// TIA Portal V18 export
// export: Created 2025-12-01T17:52:56.9110374Z, ExportSetting None, DisplayName Totally Integrated Automation Portal, DisplayVersion V18 Update 5, DisplayName TIA Portal Openness, DisplayVersion V18 Update 5, DisplayName TIA Portal Teamcenter Gateway, DisplayVersion V18, DisplayName TIA Portal Version Control Interface, DisplayVersion V18, DisplayName STEP 7 Professional, DisplayVersion V18 Update 5, DisplayName STEP 7 Safety, DisplayVersion V18, DisplayName WinCC Professional, DisplayVersion V18 Update 5
Screen "210_Cylinder_A1"  1280x800, Number=210, Template=02ManualUnit1
  ScreenLayer "Layer_0"
    FaceplateInstance "Cylinder_S71500_TP700_1" at 0,85 size 1279x80  FaceplateTypeName=03 FunctionBlocks@$@101 Cylinder@$@101.2 HMI@$@S7-1500@$@Cylinder_S71500_TP700 V 0.0.29
      Cy := STxxxCylinder001
      CylinderName := Cyl name
      HomeButtonName := Cyl go home button
      WorkButtonName := Cyl go work button
      HomeQaddress := Cyl home Q
      HomeIaddress := Cyl home I
      WorkIaddress := Cyl work I
      WorkQaddress := Cyl work Q
    FaceplateInstance "Cylinder_S71500_TP700_3" at 0,160 size 1279x80  FaceplateTypeName=03 FunctionBlocks@$@101 Cylinder@$@101.2 HMI@$@S7-1500@$@Cylinder_S71500_TP700 V 0.0.29
      Cy := STxxxCylinder002
      CylinderName := Cyl name
      HomeButtonName := Cyl go home button
      WorkButtonName := Cyl go work button
      HomeQaddress := Cyl home Q
      HomeIaddress := Cyl home I
      WorkIaddress := Cyl work I
      WorkQaddress := Cyl work Q
    Button "btnMenu4" at 384,725 size 128x75  TextOff="A-伺服 381A1 / A-Servo 381A1", TextOn="A-伺服 381A1 / A-Servo 381A1"
      on Click: ActivateScreen(Screen name := 212-Servo_381A1, Object number := 0)
    Button "btnMenu5" at 512,725 size 128x75  TextOff="A-读码器 801A1 / A-CodeReader 801A1", TextOn="A-读码器 801A1 / A-CodeReader 801A1"
      on Click: ActivateScreen(Screen name := 213 Scanner_801A1, Object number := 0)
    Button "btnMenu6" at 640,725 size 128x75  TextOff="A-读码器 804A1 / A-CodeReader 804A1", TextOn="A-读码器 804A1 / A-CodeReader 804A1"
      on Click: ActivateScreen(Screen name := 214 Scanner_804A1, Object number := 0)
    Button "btnMenu7" at 896,725 size 128x75
    Button "btnMenu6_1" at 768,725 size 128x75  TextOff="A-读码器 800A1 / A-CodeReader 800A1", TextOn="A-读码器 800A1 / A-CodeReader 800A1"
      on Click: ActivateScreen(Screen name := 215 X80Scanner_800A1, Object number := 0)
    Button "btnMenu7_1" at 1024,725 size 128x75  TextOff="下一页 / NextPage", TextOn="下一页 / NextPage"
      on Click: ActivateScreen(Screen name := 216_Cylinder_A2, Object number := 0)
    Button "按钮_9" at 128,725 size 128x75  PictureOff=向右箭头_0, TextOff="A-气缸1 / A-Cylinder1", TextOn="A-气缸1 / A-Cylinder1"
      on Click: ActivateScreen(Screen name := , Object number := 0)
    Button "btnMenu4_1" at 256,725 size 128x75  TextOff="A-伺服 380A1 / A-Servo 380A1", TextOn="A-伺服 380A1 / A-Servo 380A1"
      on Click: ActivateScreen(Screen name := 211-Servo_380A1, Object number := 0)
    GraphicView "图形视图_1" at 305,251 size 656x434  Picture=图形_46
